// TwinCAT 3 PLC project plc01
// ProgramVersion: 3.1.4023.0
// libraries:
//   Tc2_Standard, * (Beckhoff Automation GmbH)
//   Tc2_System, * (Beckhoff Automation GmbH)
//   Tc3_Module, * (Beckhoff Automation GmbH)
// project tree:
//   / PlcTask.TcTTO
//   POUs/ MAIN.TcPOU
// real-time tasks:
//   TASK PlcTask: cycle T#10ms, priority 20, ADS port 350

CONFIGURATION plc01
    RESOURCE PLC ON TwinCAT3
        TASK PlcTask(INTERVAL := T#10ms, PRIORITY := 20);
        PROGRAM MAIN WITH PlcTask : MAIN;
    END_RESOURCE
END_CONFIGURATION

// ---- POUs/MAIN.TcPOU
PROGRAM MAIN
VAR
	bInit: BOOL;
	sStart: STRING;
END_VAR

//Develolep BY Kauê Koschitz Roratto
//https://github.com/KaueKoschitzRoratto
//https://www.linkedin.com/in/kauekoschitzroratto/
//kaue.roratto@outlook.com.br

IF bInit THEN
	sStart:= 'project Started';
END_IF

END_PROGRAM
